(* IEC 61131-3 sources: CodesysTest/alpha/export/FBs/Components/MotorizedSealFlattenersFB_BagFeed.pou/Mode.prop, 1 file *)

(* ---- Set.pm.st ---- *)
(*#-#-#-#-#-#-#-#-#-#---Declaration---#-#-#-#-#-#-#-#-#-#-#-#-#*)

VAR
END_VAR
(*#-#-#-#-#-#-#-#-#-#---Implementation---#-#-#-#-#-#-#-#-#-#-#-#-#*)

_mode := Mode;
